// TIA Portal project "GR36_BP_PSElevator" (V17)

(* hardware
DEVICE "ET 200SP station_1"  ET 200SP-Station
   slot 0: "Rack_0"  Rack  6ES5 710-8MAx1
   slot 1: "PLC_1"  CPU 1510SP-1 PN  6ES7 510-1DJ01-0AB0  V2.1
      slot 32768: "PROFINET interface_1"  X1
   slot 2: "DI 8x24VDC HF_1"  DI 8x24VDC HF  6ES7 131-6BF00-0CA0  V2.0
      slot 1: "DI 8x24VDC HF_1"  DI 8x24VDC HF
   slot 3: "DI 8x24VDC BA_1"  DI 8x24VDC BA  6ES7 131-6BF00-0AA0  V1.0
      slot 1: "DI 8x24VDC BA_1"  DI 8x24VDC BA
   slot 4: "DQ 8x24VDC/0.5A ST_1"  DQ 8x24VDC/0.5A ST  6ES7 132-6BF00-0BA0  V1.1
      slot 1: "DQ 8x24VDC/0.5A ST_1"  DQ 8x24VDC/0.5A ST
   slot 5: "AI 2xU/I 2-,4-wire HF_1"  AI 2xU/I 2-,4-wire HF  6ES7 134-6HB00-0CA1  V2.0
      slot 1: "AI 2xU/I 2-,4-wire HF_1"  AI 2xU/I 2-,4-wire HF
   slot 6: "Server module_1"  Server module  6ES7 193-6PA00-0AA0  V1.1
      slot 1: "Server module_1"  Server module
   slot 127: "BA 2xRJ45"  BA 2xRJ45  6ES7 193-6AR00-0AA0  V0.0
      slot 32769: "Port_1"  X1 P1  6ES7 193-6AR00-0AA0
      slot 32770: "Port_2"  X1 P2  6ES7 193-6AR00-0AA0
*)

// ===== PLC "PLC_1"  CPU 1510SP-1 PN =====

VAR_GLOBAL   // PLC tag table "Default tag table"
   "System_Byte" AT %MB70 : Byte;
   "FirstScan" AT %M70.0 : Bool;
   "DiagStatusUpdate" AT %M70.1 : Bool;
   "AlwaysTRUE" AT %M70.2 : Bool;
   "AlwaysFALSE" AT %M70.3 : Bool;
   "Clock_Byte" AT %MB69 : Byte;
   "Clock_10Hz" AT %M69.0 : Bool;
   "Clock_5Hz" AT %M69.1 : Bool;
   "Clock_2.5Hz" AT %M69.2 : Bool;
   "Clock_2Hz" AT %M69.3 : Bool;
   "Clock_1.25Hz" AT %M69.4 : Bool;
   "Clock_1Hz" AT %M69.5 : Bool;
   "Clock_0.625Hz" AT %M69.6 : Bool;
   "Clock_0.5Hz" AT %M69.7 : Bool;
END_VAR

VAR_GLOBAL   // PLC tag table "PLC_dq"
   "dq_LedGreen" AT %Q204.0 : Bool;
   "dq_LedRed" AT %Q204.1 : Bool;
   "dq_LedWhite" AT %Q204.2 : Bool;
   "dq_LedBlue" AT %Q204.3 : Bool;
END_VAR

VAR_GLOBAL   // PLC tag table "PLC_di"
   "di_StartButton" AT %I202.0 : Bool;
   "di_StopButton" AT %I202.1 : Bool;
   "di_Selector" AT %I202.2 : Bool;
   "di_Reset" AT %I202.3 : Bool;
   "di_SwitchForward" AT %I201.0 : Bool;
   "di_SwitchBackward" AT %I201.1 : Bool;
   "di_SwitchBay1" AT %I201.2 : Bool;
   "di_SwitchBay2" AT %I201.3 : Bool;
END_VAR

VAR_GLOBAL   // PLC tag table "FactoryIO_dq"
   "dq_M1" AT %Q7.0 : Bool;
   "dq_M2" AT %Q7.1 : Bool;
   "dq_M3" AT %Q7.2 : Bool;
   "dq_Turntable_1_Turn" AT %Q7.3 : Bool;
   "dq_Turntable_1_Roll+" AT %Q7.4 : Bool;
   "dq_Turntable_1_Roll-" AT %Q7.5 : Bool;
   "dq_Elevator_1_Up" AT %Q8.0 : Bool;
   "dq_Elevator_1_Down" AT %Q8.1 : Bool;
   "dq_Elevator_1_Slow" AT %Q8.2 : Bool;
   "dq_M5" AT %Q8.3 : Bool;
   "dq_M6" AT %Q8.4 : Bool;
   "dq_M4_Elevator_1_+" AT %Q7.6 : Bool;
   "dq_M4_Elevator_1_-" AT %Q7.7 : Bool;
END_VAR

VAR_GLOBAL   // PLC tag table "FactoryIO_di"
   "di_B1" AT %I7.0 : Bool;
   "di_B3_Exit" AT %I7.1 : Bool;
   "di_B5_Exit" AT %I7.2 : Bool;
   "di_B6_Exit" AT %I7.3 : Bool;
   "di_B3_Entry" AT %I7.4 : Bool;
   "di_B5_Entry" AT %I7.5 : Bool;
   "di_B6_Entry" AT %I7.6 : Bool;
   "di_Elevator_1_LeftLimit" AT %I7.7 : Bool;
   "di_Elevator_1_RightLimit" AT %I8.0 : Bool;
   "di_HightSensor_Lift_0" AT %I8.1 : Bool;
   "di_HightSensor_Lift_1" AT %I8.2 : Bool;
   "di_LowSensor_Lift_0" AT %I8.3 : Bool;
   "di_LowSensor_Lift_1" AT %I8.4 : Bool;
   "di_M3_Encoder_Signal_A" AT %I8.5 : Bool;
   "di_M3_Encoder_Signal_B" AT %I8.6 : Bool;
   "di_Turntable_1_Limit_0" AT %I8.7 : Bool;
   "di_Turntable_1_Limit_90" AT %I9.0 : Bool;
   "di_Turntable_1_BackLimit" AT %I9.1 : Bool;
   "di_Turntable_1_FrontLimit" AT %I9.2 : Bool;
   "di_FactoryIO_Running" AT %I9.7 : Bool;
END_VAR

TYPE "edge_detection"
   STRUCT
      OneShoot_Positive : Bool;
      OneShoot_Negative : Bool;
      memory : Struct
         PreviousState_Positive : Bool;
         PreviousState_Negative : Bool;
      END_STRUCT;
   END_STRUCT;
END_TYPE

DATA_BLOCK "db_output"   // DB1
{ S7_Optimized_Access := 'TRUE' }
VERSION : 0.1
   VAR
      M1_Auto_Forward : Bool;
      M2_Auto_Forward : Bool;
      M3_Auto_Forward : Bool;
      "turntable_1_roll_Auto_-" : Bool;
      "turntable_1_roll_Auto_+" : Bool;
      "M4_elevator_1_Auto_+" : Bool;
      "M4_elevator_1_Auto_-" : Bool;
      elevator_1_Auto_Up : Bool;
      elevator_1_Auto_Down : Bool;
      elevator_1_Auto_Slow : Bool;
      M6_Auto_Forward : Bool;
   END_VAR
BEGIN
END_DATA_BLOCK

DATA_BLOCK "db_turntable"   // DB2
{ S7_Optimized_Access := 'TRUE' }
VERSION : 0.1
   VAR
      isOccupied : Bool;
      isM1PackageReady : Bool;
      isM2PackageReady : Bool;
      isM1PackageTransported2Turntable : Bool;
   END_VAR
BEGIN
END_DATA_BLOCK

DATA_BLOCK "db_mode"   // DB3
{ S7_Optimized_Access := 'TRUE' }
VERSION : 0.1
   VAR
      GlobalError : Bool;
      Auto : Bool;
   END_VAR
BEGIN
END_DATA_BLOCK

DATA_BLOCK "db_error"   // DB4
{ S7_Optimized_Access := 'TRUE' }
VERSION : 0.1
   VAR
      er_1 : Bool;
   END_VAR
BEGIN
END_DATA_BLOCK

DATA_BLOCK "db_edge"   // DB5
{ S7_Optimized_Access := 'TRUE' }
VERSION : 0.1
   VAR
      Elevator_1_RightLimit : "edge_detection";
      Elevator_1_LeftLimit : "edge_detection";
      B1 : "edge_detection";
      Turntable_1_BackLimit : "edge_detection";
      Turntable_1_FrontLimit : "edge_detection";
      B3_Entry : "edge_detection";
      B3_End : "edge_detection";
      Lift_1_Height : "edge_detection";
      Lift_1_Low : "edge_detection";
      Lift_0_Height : "edge_detection";
      Lift_0_Low : "edge_detection";
      B6_Entry : "edge_detection";
      B6_Exit : "edge_detection";
      B3_Exit : "edge_detection";
   END_VAR
BEGIN
END_DATA_BLOCK

DATA_BLOCK "db_settings"   // DB6
{ S7_Optimized_Access := 'TRUE' }
VERSION : 0.1
   VAR RETAIN
      M1_ReadyDelay : Time := t#5s;
      M2_ReadyDelay : Time := t#5s;
   END_VAR
BEGIN
END_DATA_BLOCK

DATA_BLOCK "db_elevator"   // DB7
{ S7_Optimized_Access := 'TRUE' }
VERSION : 0.1
   VAR
      isOccupied : Bool;
      slowMode : Bool;
      isLineB3Occupied : Bool;
   END_VAR
BEGIN
END_DATA_BLOCK

FUNCTION "fc_output" : Void   // FC1, LAD
{ S7_Optimized_Access := 'TRUE' }
VERSION : 0.1
BEGIN

REGION Network 1: M1
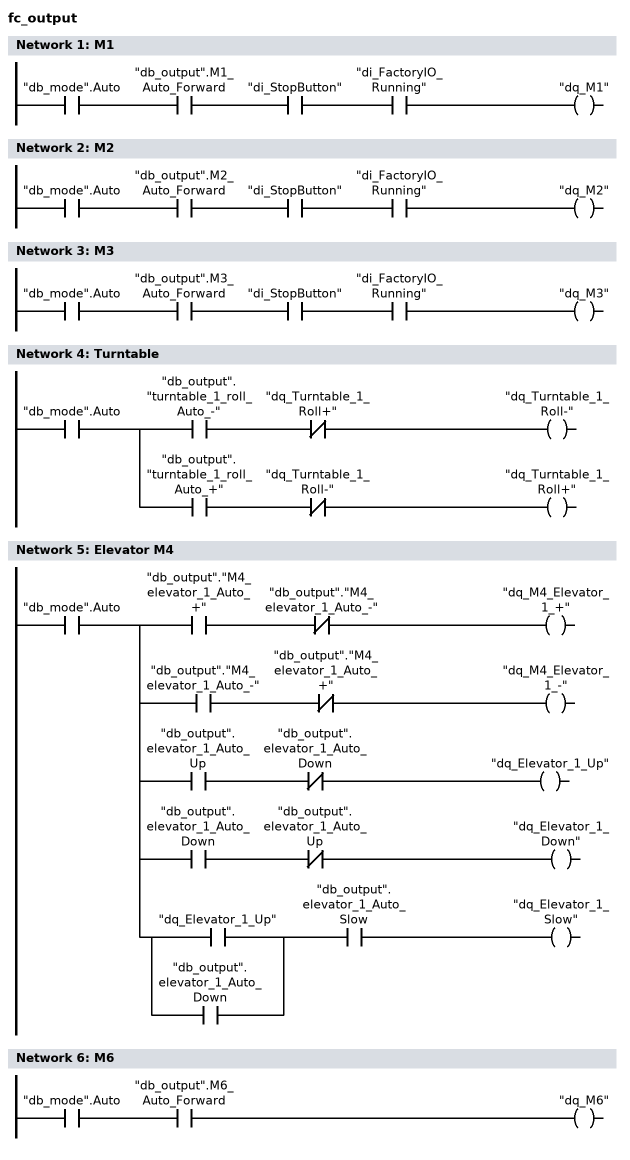
   RUNG wire#powerrail
      Contact( "db_mode".Auto )
      Contact( "db_output".M1_Auto_Forward )
      Contact( "di_StopButton" )
      Contact( "di_FactoryIO_Running" )
      Coil( "dq_M1" )
   END_RUNG
   // the same network as SCL:
   "dq_M1" := "db_mode".Auto AND "db_output".M1_Auto_Forward AND "di_StopButton" AND "di_FactoryIO_Running";
END_REGION

REGION Network 2: M2
   RUNG wire#powerrail
      Contact( "db_mode".Auto )
      Contact( "db_output".M2_Auto_Forward )
      Contact( "di_StopButton" )
      Contact( "di_FactoryIO_Running" )
      Coil( "dq_M2" )
   END_RUNG
   // the same network as SCL:
   "dq_M2" := "db_mode".Auto AND "db_output".M2_Auto_Forward AND "di_StopButton" AND "di_FactoryIO_Running";
END_REGION

REGION Network 3: M3
   RUNG wire#powerrail
      Contact( "db_mode".Auto )
      Contact( "db_output".M3_Auto_Forward )
      Contact( "di_StopButton" )
      Contact( "di_FactoryIO_Running" )
      Coil( "dq_M3" )
   END_RUNG
   // the same network as SCL:
   "dq_M3" := "db_mode".Auto AND "db_output".M3_Auto_Forward AND "di_StopButton" AND "di_FactoryIO_Running";
END_REGION

REGION Network 4: Turntable
   RUNG wire#powerrail
      Contact( "db_mode".Auto )
      wire#w1
      Contact( "db_output"."turntable_1_roll_Auto_-" )
      I_Contact( "dq_Turntable_1_Roll+" )
      Coil( "dq_Turntable_1_Roll-" )
   END_RUNG
   RUNG wire#w1
      Contact( "db_output"."turntable_1_roll_Auto_+" )
      I_Contact( "dq_Turntable_1_Roll-" )
      Coil( "dq_Turntable_1_Roll+" )
   END_RUNG
   // the same network as SCL:
   "dq_Turntable_1_Roll-" := "db_mode".Auto AND "db_output"."turntable_1_roll_Auto_-" AND NOT "dq_Turntable_1_Roll+";
   "dq_Turntable_1_Roll+" := "db_mode".Auto AND "db_output"."turntable_1_roll_Auto_+" AND NOT "dq_Turntable_1_Roll-";
END_REGION

REGION Network 5: Elevator M4
   RUNG wire#powerrail
      Contact( "db_mode".Auto )
      wire#w1
      Contact( "db_output"."M4_elevator_1_Auto_+" )
      I_Contact( "db_output"."M4_elevator_1_Auto_-" )
      Coil( "dq_M4_Elevator_1_+" )
   END_RUNG
   RUNG wire#w1
      Contact( "db_output"."M4_elevator_1_Auto_-" )
      I_Contact( "db_output"."M4_elevator_1_Auto_+" )
      Coil( "dq_M4_Elevator_1_-" )
   END_RUNG
   RUNG wire#w1
      Contact( "db_output".elevator_1_Auto_Up )
      I_Contact( "db_output".elevator_1_Auto_Down )
      Coil( "dq_Elevator_1_Up" )
   END_RUNG
   RUNG wire#w1
      Contact( "db_output".elevator_1_Auto_Down )
      I_Contact( "db_output".elevator_1_Auto_Up )
      Coil( "dq_Elevator_1_Down" )
   END_RUNG
   RUNG wire#w1
      Contact( "dq_Elevator_1_Up" )
      wire#w2
      Contact( "db_output".elevator_1_Auto_Slow )
      Coil( "dq_Elevator_1_Slow" )
   END_RUNG
   RUNG wire#w1
      Contact( "db_output".elevator_1_Auto_Down )
   END_RUNG wire#w2
   // the same network as SCL:
   "dq_M4_Elevator_1_+" := "db_mode".Auto AND "db_output"."M4_elevator_1_Auto_+" AND NOT "db_output"."M4_elevator_1_Auto_-";
   "dq_M4_Elevator_1_-" := "db_mode".Auto AND "db_output"."M4_elevator_1_Auto_-" AND NOT "db_output"."M4_elevator_1_Auto_+";
   "dq_Elevator_1_Up" := "db_mode".Auto AND "db_output".elevator_1_Auto_Up AND NOT "db_output".elevator_1_Auto_Down;
   "dq_Elevator_1_Down" := "db_mode".Auto AND "db_output".elevator_1_Auto_Down AND NOT "db_output".elevator_1_Auto_Up;
   "dq_Elevator_1_Slow" := "db_mode".Auto AND ("dq_Elevator_1_Up" OR "db_output".elevator_1_Auto_Down) AND "db_output".elevator_1_Auto_Slow;
END_REGION

REGION Network 6: M6
   RUNG wire#powerrail
      Contact( "db_mode".Auto )
      Contact( "db_output".M6_Auto_Forward )
      Coil( "dq_M6" )
   END_RUNG
   // the same network as SCL:
   "dq_M6" := "db_mode".Auto AND "db_output".M6_Auto_Forward;
END_REGION
END_FUNCTION

FUNCTION "fc_mode" : Void   // FC2, LAD
{ S7_Optimized_Access := 'TRUE' }
VERSION : 0.1
BEGIN

REGION Network 1: Set auto mode
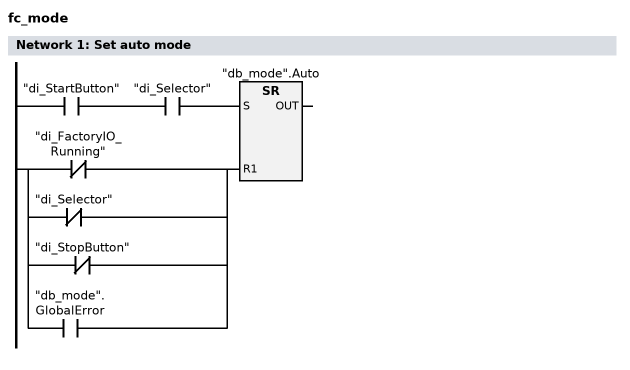
   RUNG wire#powerrail
      Contact( "di_StartButton" )
      Contact( "di_Selector" )
      S_SR(operand := "db_mode".Auto, r1 := wire#w1)
   END_RUNG
   RUNG wire#powerrail
      I_Contact( "di_FactoryIO_Running" )
   END_RUNG wire#w1
   RUNG wire#powerrail
      I_Contact( "di_Selector" )
   END_RUNG wire#w1
   RUNG wire#powerrail
      I_Contact( "di_StopButton" )
   END_RUNG wire#w1
   RUNG wire#powerrail
      Contact( "db_mode".GlobalError )
   END_RUNG wire#w1
   // the same network as SCL:
   IF "di_StartButton" AND "di_Selector" THEN
       "db_mode".Auto := TRUE;   // SR flip-flop
   END_IF;
   IF NOT "di_FactoryIO_Running" OR NOT "di_Selector" OR NOT "di_StopButton" OR "db_mode".GlobalError THEN
       "db_mode".Auto := FALSE;
   END_IF;
END_REGION
END_FUNCTION

FUNCTION "fc_auto" : Void   // FC3, LAD
{ S7_Optimized_Access := 'TRUE' }
VERSION : 0.1
BEGIN

REGION Network 1: M1 Transport the package to the turntable if the turntable is not occupied
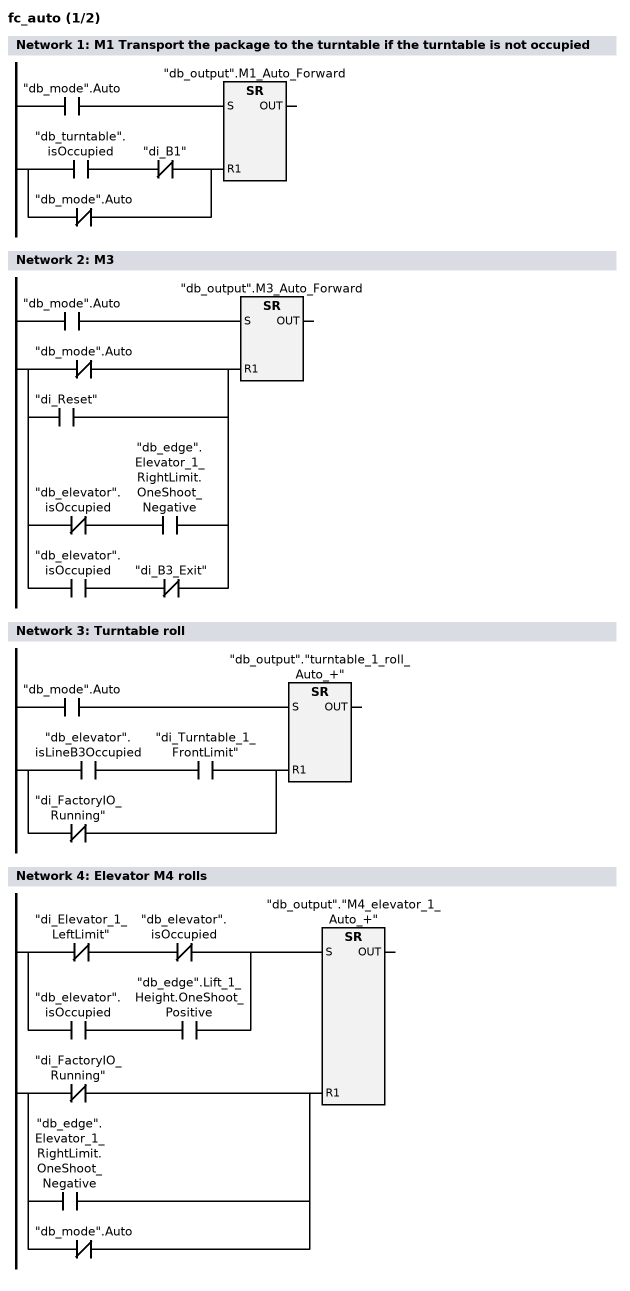
   RUNG wire#powerrail
      Contact( "db_mode".Auto )
      S_SR(operand := "db_output".M1_Auto_Forward, r1 := wire#w1)
   END_RUNG
   RUNG wire#powerrail
      Contact( "db_turntable".isOccupied )
      I_Contact( "di_B1" )
   END_RUNG wire#w1
   RUNG wire#powerrail
      I_Contact( "db_mode".Auto )
   END_RUNG wire#w1
   // the same network as SCL:
   IF "db_mode".Auto THEN
       "db_output".M1_Auto_Forward := TRUE;   // SR flip-flop
   END_IF;
   IF ("db_turntable".isOccupied AND NOT "di_B1") OR NOT "db_mode".Auto THEN
       "db_output".M1_Auto_Forward := FALSE;
   END_IF;
END_REGION

REGION Network 2: M3
   RUNG wire#powerrail
      Contact( "db_mode".Auto )
      S_SR(operand := "db_output".M3_Auto_Forward, r1 := wire#w1)
   END_RUNG
   RUNG wire#powerrail
      I_Contact( "db_mode".Auto )
   END_RUNG wire#w1
   RUNG wire#powerrail
      Contact( "di_Reset" )
   END_RUNG wire#w1
   RUNG wire#powerrail
      I_Contact( "db_elevator".isOccupied )
      Contact( "db_edge".Elevator_1_RightLimit.OneShoot_Negative )
   END_RUNG wire#w1
   RUNG wire#powerrail
      Contact( "db_elevator".isOccupied )
      I_Contact( "di_B3_Exit" )
   END_RUNG wire#w1
   // the same network as SCL:
   IF "db_mode".Auto THEN
       "db_output".M3_Auto_Forward := TRUE;   // SR flip-flop
   END_IF;
   IF NOT "db_mode".Auto OR "di_Reset" OR (NOT "db_elevator".isOccupied AND "db_edge".Elevator_1_RightLimit.OneShoot_Negative) OR ("db_elevator".isOccupied AND NOT "di_B3_Exit") THEN
       "db_output".M3_Auto_Forward := FALSE;
   END_IF;
END_REGION

REGION Network 3: Turntable roll
   RUNG wire#powerrail
      Contact( "db_mode".Auto )
      S_SR(operand := "db_output"."turntable_1_roll_Auto_+", r1 := wire#w1)
   END_RUNG
   RUNG wire#powerrail
      Contact( "db_elevator".isLineB3Occupied )
      Contact( "di_Turntable_1_FrontLimit" )
   END_RUNG wire#w1
   RUNG wire#powerrail
      I_Contact( "di_FactoryIO_Running" )
   END_RUNG wire#w1
   // the same network as SCL:
   IF "db_mode".Auto THEN
       "db_output"."turntable_1_roll_Auto_+" := TRUE;   // SR flip-flop
   END_IF;
   IF ("db_elevator".isLineB3Occupied AND "di_Turntable_1_FrontLimit") OR NOT "di_FactoryIO_Running" THEN
       "db_output"."turntable_1_roll_Auto_+" := FALSE;
   END_IF;
END_REGION

REGION Network 4: Elevator M4 rolls
   RUNG wire#powerrail
      I_Contact( "di_Elevator_1_LeftLimit" )
      I_Contact( "db_elevator".isOccupied )
      wire#w1
      S_SR(operand := "db_output"."M4_elevator_1_Auto_+", r1 := wire#w2)
   END_RUNG
   RUNG wire#powerrail
      Contact( "db_elevator".isOccupied )
      Contact( "db_edge".Lift_1_Height.OneShoot_Positive )
   END_RUNG wire#w1
   RUNG wire#powerrail
      I_Contact( "di_FactoryIO_Running" )
   END_RUNG wire#w2
   RUNG wire#powerrail
      Contact( "db_edge".Elevator_1_RightLimit.OneShoot_Negative )
   END_RUNG wire#w2
   RUNG wire#powerrail
      I_Contact( "db_mode".Auto )
   END_RUNG wire#w2
   // the same network as SCL:
   IF (NOT "di_Elevator_1_LeftLimit" AND NOT "db_elevator".isOccupied) OR ("db_elevator".isOccupied AND "db_edge".Lift_1_Height.OneShoot_Positive) THEN
       "db_output"."M4_elevator_1_Auto_+" := TRUE;   // SR flip-flop
   END_IF;
   IF NOT "di_FactoryIO_Running" OR "db_edge".Elevator_1_RightLimit.OneShoot_Negative OR NOT "db_mode".Auto THEN
       "db_output"."M4_elevator_1_Auto_+" := FALSE;
   END_IF;
END_REGION

REGION Network 5: Elevator lift
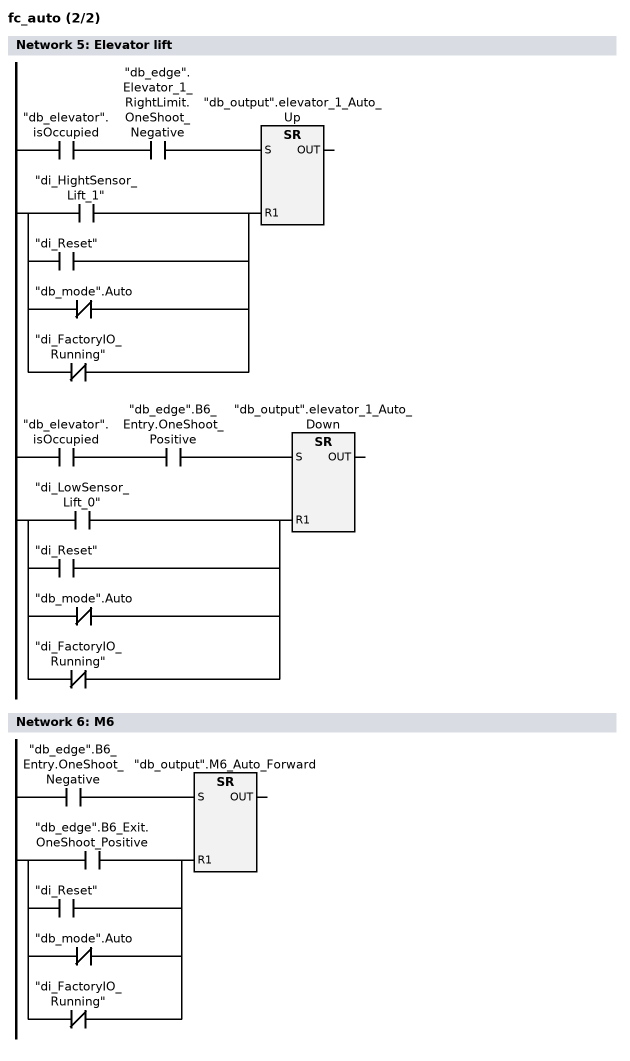
   RUNG wire#powerrail
      Contact( "db_elevator".isOccupied )
      Contact( "db_edge".Elevator_1_RightLimit.OneShoot_Negative )
      S_SR(operand := "db_output".elevator_1_Auto_Up, r1 := wire#w1)
   END_RUNG
   RUNG wire#powerrail
      Contact( "di_HightSensor_Lift_1" )
   END_RUNG wire#w1
   RUNG wire#powerrail
      Contact( "di_Reset" )
   END_RUNG wire#w1
   RUNG wire#powerrail
      I_Contact( "db_mode".Auto )
   END_RUNG wire#w1
   RUNG wire#powerrail
      I_Contact( "di_FactoryIO_Running" )
   END_RUNG wire#w1
   RUNG wire#powerrail
      Contact( "db_elevator".isOccupied )
      Contact( "db_edge".B6_Entry.OneShoot_Positive )
      S_SR(operand := "db_output".elevator_1_Auto_Down, r1 := wire#w2)
   END_RUNG
   RUNG wire#powerrail
      Contact( "di_LowSensor_Lift_0" )
   END_RUNG wire#w2
   RUNG wire#powerrail
      Contact( "di_Reset" )
   END_RUNG wire#w2
   RUNG wire#powerrail
      I_Contact( "db_mode".Auto )
   END_RUNG wire#w2
   RUNG wire#powerrail
      I_Contact( "di_FactoryIO_Running" )
   END_RUNG wire#w2
   // the same network as SCL:
   IF "db_elevator".isOccupied AND "db_edge".Elevator_1_RightLimit.OneShoot_Negative THEN
       "db_output".elevator_1_Auto_Up := TRUE;   // SR flip-flop
   END_IF;
   IF "di_HightSensor_Lift_1" OR "di_Reset" OR NOT "db_mode".Auto OR NOT "di_FactoryIO_Running" THEN
       "db_output".elevator_1_Auto_Up := FALSE;
   END_IF;
   IF "db_elevator".isOccupied AND "db_edge".B6_Entry.OneShoot_Positive THEN
       "db_output".elevator_1_Auto_Down := TRUE;   // SR flip-flop
   END_IF;
   IF "di_LowSensor_Lift_0" OR "di_Reset" OR NOT "db_mode".Auto OR NOT "di_FactoryIO_Running" THEN
       "db_output".elevator_1_Auto_Down := FALSE;
   END_IF;
END_REGION

REGION Network 6: M6
   RUNG wire#powerrail
      Contact( "db_edge".B6_Entry.OneShoot_Negative )
      S_SR(operand := "db_output".M6_Auto_Forward, r1 := wire#w1)
   END_RUNG
   RUNG wire#powerrail
      Contact( "db_edge".B6_Exit.OneShoot_Positive )
   END_RUNG wire#w1
   RUNG wire#powerrail
      Contact( "di_Reset" )
   END_RUNG wire#w1
   RUNG wire#powerrail
      I_Contact( "db_mode".Auto )
   END_RUNG wire#w1
   RUNG wire#powerrail
      I_Contact( "di_FactoryIO_Running" )
   END_RUNG wire#w1
   // the same network as SCL:
   IF "db_edge".B6_Entry.OneShoot_Negative THEN
       "db_output".M6_Auto_Forward := TRUE;   // SR flip-flop
   END_IF;
   IF "db_edge".B6_Exit.OneShoot_Positive OR "di_Reset" OR NOT "db_mode".Auto OR NOT "di_FactoryIO_Running" THEN
       "db_output".M6_Auto_Forward := FALSE;
   END_IF;
END_REGION
END_FUNCTION

FUNCTION "fc_turntable" : Void   // FC4, LAD
{ S7_Optimized_Access := 'TRUE' }
VERSION : 0.1
BEGIN

REGION Network 1: Set when turn table is occupied
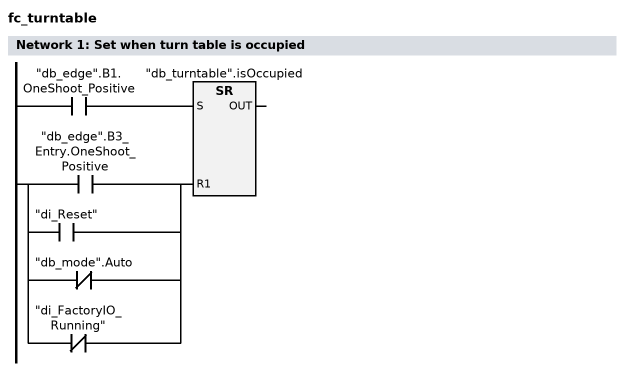
   RUNG wire#powerrail
      Contact( "db_edge".B1.OneShoot_Positive )
      S_SR(operand := "db_turntable".isOccupied, r1 := wire#w1)
   END_RUNG
   RUNG wire#powerrail
      Contact( "db_edge".B3_Entry.OneShoot_Positive )
   END_RUNG wire#w1
   RUNG wire#powerrail
      Contact( "di_Reset" )
   END_RUNG wire#w1
   RUNG wire#powerrail
      I_Contact( "db_mode".Auto )
   END_RUNG wire#w1
   RUNG wire#powerrail
      I_Contact( "di_FactoryIO_Running" )
   END_RUNG wire#w1
   // the same network as SCL:
   IF "db_edge".B1.OneShoot_Positive THEN
       "db_turntable".isOccupied := TRUE;   // SR flip-flop
   END_IF;
   IF "db_edge".B3_Entry.OneShoot_Positive OR "di_Reset" OR NOT "db_mode".Auto OR NOT "di_FactoryIO_Running" THEN
       "db_turntable".isOccupied := FALSE;
   END_IF;
END_REGION
END_FUNCTION

FUNCTION "fc_edge" : Void   // FC5, LAD
{ S7_Optimized_Access := 'TRUE' }
VERSION : 0.1
   VAR_TEMP   // added for the SCL form of the ladder/FBD networks
      _w1 : Bool;
      _w2 : Bool;
      _w3 : Bool;
      _w4 : Bool;
   END_VAR
BEGIN

REGION Network 1: Turntable 1
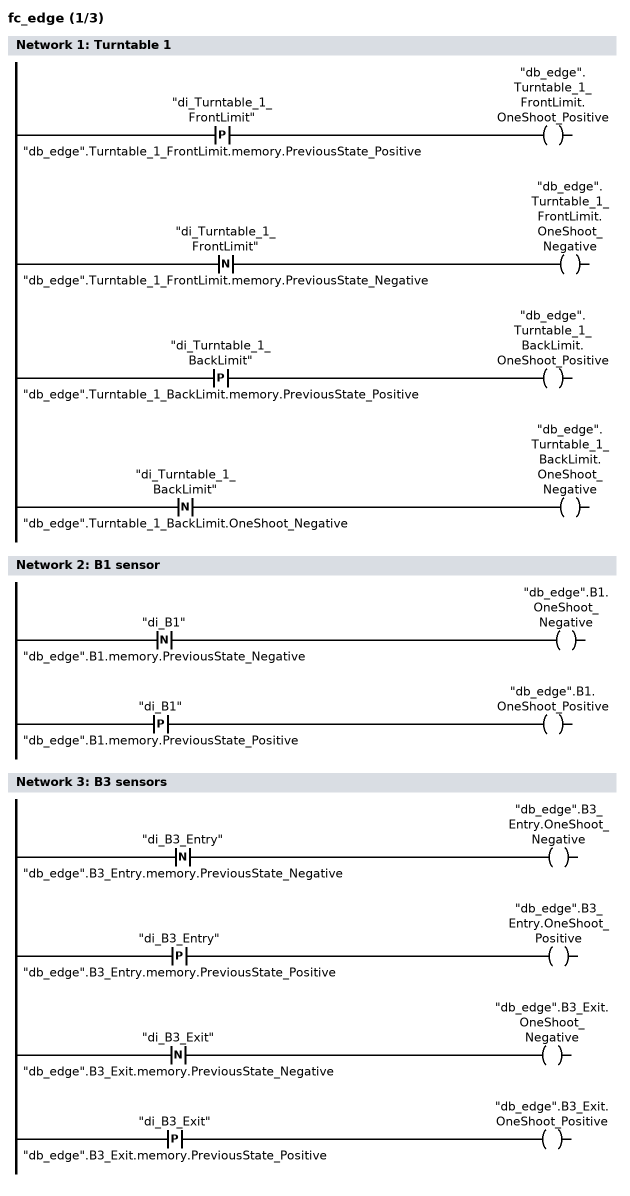
   RUNG wire#powerrail
      P_Contact(operand := "di_Turntable_1_FrontLimit", bit := "db_edge".Turntable_1_FrontLimit.memory.PreviousState_Positive)
      Coil( "db_edge".Turntable_1_FrontLimit.OneShoot_Positive )
   END_RUNG
   RUNG wire#powerrail
      N_Contact(operand := "di_Turntable_1_FrontLimit", bit := "db_edge".Turntable_1_FrontLimit.memory.PreviousState_Negative)
      Coil( "db_edge".Turntable_1_FrontLimit.OneShoot_Negative )
   END_RUNG
   RUNG wire#powerrail
      P_Contact(operand := "di_Turntable_1_BackLimit", bit := "db_edge".Turntable_1_BackLimit.memory.PreviousState_Positive)
      Coil( "db_edge".Turntable_1_BackLimit.OneShoot_Positive )
   END_RUNG
   RUNG wire#powerrail
      N_Contact(operand := "di_Turntable_1_BackLimit", bit := "db_edge".Turntable_1_BackLimit.OneShoot_Negative)
      Coil( "db_edge".Turntable_1_BackLimit.OneShoot_Negative )
   END_RUNG
   // the same network as SCL:
   #_w1 := "di_Turntable_1_FrontLimit" AND NOT "db_edge".Turntable_1_FrontLimit.memory.PreviousState_Positive;   // rising edge of "di_Turntable_1_FrontLimit"
   "db_edge".Turntable_1_FrontLimit.memory.PreviousState_Positive := "di_Turntable_1_FrontLimit";
   "db_edge".Turntable_1_FrontLimit.OneShoot_Positive := #_w1;
   #_w2 := NOT "di_Turntable_1_FrontLimit" AND "db_edge".Turntable_1_FrontLimit.memory.PreviousState_Negative;   // falling edge of "di_Turntable_1_FrontLimit"
   "db_edge".Turntable_1_FrontLimit.memory.PreviousState_Negative := "di_Turntable_1_FrontLimit";
   "db_edge".Turntable_1_FrontLimit.OneShoot_Negative := #_w2;
   #_w3 := "di_Turntable_1_BackLimit" AND NOT "db_edge".Turntable_1_BackLimit.memory.PreviousState_Positive;   // rising edge of "di_Turntable_1_BackLimit"
   "db_edge".Turntable_1_BackLimit.memory.PreviousState_Positive := "di_Turntable_1_BackLimit";
   "db_edge".Turntable_1_BackLimit.OneShoot_Positive := #_w3;
   #_w4 := NOT "di_Turntable_1_BackLimit" AND "db_edge".Turntable_1_BackLimit.OneShoot_Negative;   // falling edge of "di_Turntable_1_BackLimit"
   "db_edge".Turntable_1_BackLimit.OneShoot_Negative := "di_Turntable_1_BackLimit";
   "db_edge".Turntable_1_BackLimit.OneShoot_Negative := #_w4;
END_REGION

REGION Network 2: B1 sensor
   RUNG wire#powerrail
      N_Contact(operand := "di_B1", bit := "db_edge".B1.memory.PreviousState_Negative)
      Coil( "db_edge".B1.OneShoot_Negative )
   END_RUNG
   RUNG wire#powerrail
      P_Contact(operand := "di_B1", bit := "db_edge".B1.memory.PreviousState_Positive)
      Coil( "db_edge".B1.OneShoot_Positive )
   END_RUNG
   // the same network as SCL:
   #_w1 := NOT "di_B1" AND "db_edge".B1.memory.PreviousState_Negative;   // falling edge of "di_B1"
   "db_edge".B1.memory.PreviousState_Negative := "di_B1";
   "db_edge".B1.OneShoot_Negative := #_w1;
   #_w2 := "di_B1" AND NOT "db_edge".B1.memory.PreviousState_Positive;   // rising edge of "di_B1"
   "db_edge".B1.memory.PreviousState_Positive := "di_B1";
   "db_edge".B1.OneShoot_Positive := #_w2;
END_REGION

REGION Network 3: B3 sensors
   RUNG wire#powerrail
      N_Contact(operand := "di_B3_Entry", bit := "db_edge".B3_Entry.memory.PreviousState_Negative)
      Coil( "db_edge".B3_Entry.OneShoot_Negative )
   END_RUNG
   RUNG wire#powerrail
      P_Contact(operand := "di_B3_Entry", bit := "db_edge".B3_Entry.memory.PreviousState_Positive)
      Coil( "db_edge".B3_Entry.OneShoot_Positive )
   END_RUNG
   RUNG wire#powerrail
      N_Contact(operand := "di_B3_Exit", bit := "db_edge".B3_Exit.memory.PreviousState_Negative)
      Coil( "db_edge".B3_Exit.OneShoot_Negative )
   END_RUNG
   RUNG wire#powerrail
      P_Contact(operand := "di_B3_Exit", bit := "db_edge".B3_Exit.memory.PreviousState_Positive)
      Coil( "db_edge".B3_Exit.OneShoot_Positive )
   END_RUNG
   // the same network as SCL:
   #_w1 := NOT "di_B3_Entry" AND "db_edge".B3_Entry.memory.PreviousState_Negative;   // falling edge of "di_B3_Entry"
   "db_edge".B3_Entry.memory.PreviousState_Negative := "di_B3_Entry";
   "db_edge".B3_Entry.OneShoot_Negative := #_w1;
   #_w2 := "di_B3_Entry" AND NOT "db_edge".B3_Entry.memory.PreviousState_Positive;   // rising edge of "di_B3_Entry"
   "db_edge".B3_Entry.memory.PreviousState_Positive := "di_B3_Entry";
   "db_edge".B3_Entry.OneShoot_Positive := #_w2;
   #_w3 := NOT "di_B3_Exit" AND "db_edge".B3_Exit.memory.PreviousState_Negative;   // falling edge of "di_B3_Exit"
   "db_edge".B3_Exit.memory.PreviousState_Negative := "di_B3_Exit";
   "db_edge".B3_Exit.OneShoot_Negative := #_w3;
   #_w4 := "di_B3_Exit" AND NOT "db_edge".B3_Exit.memory.PreviousState_Positive;   // rising edge of "di_B3_Exit"
   "db_edge".B3_Exit.memory.PreviousState_Positive := "di_B3_Exit";
   "db_edge".B3_Exit.OneShoot_Positive := #_w4;
END_REGION

REGION Network 4: Elevator 1
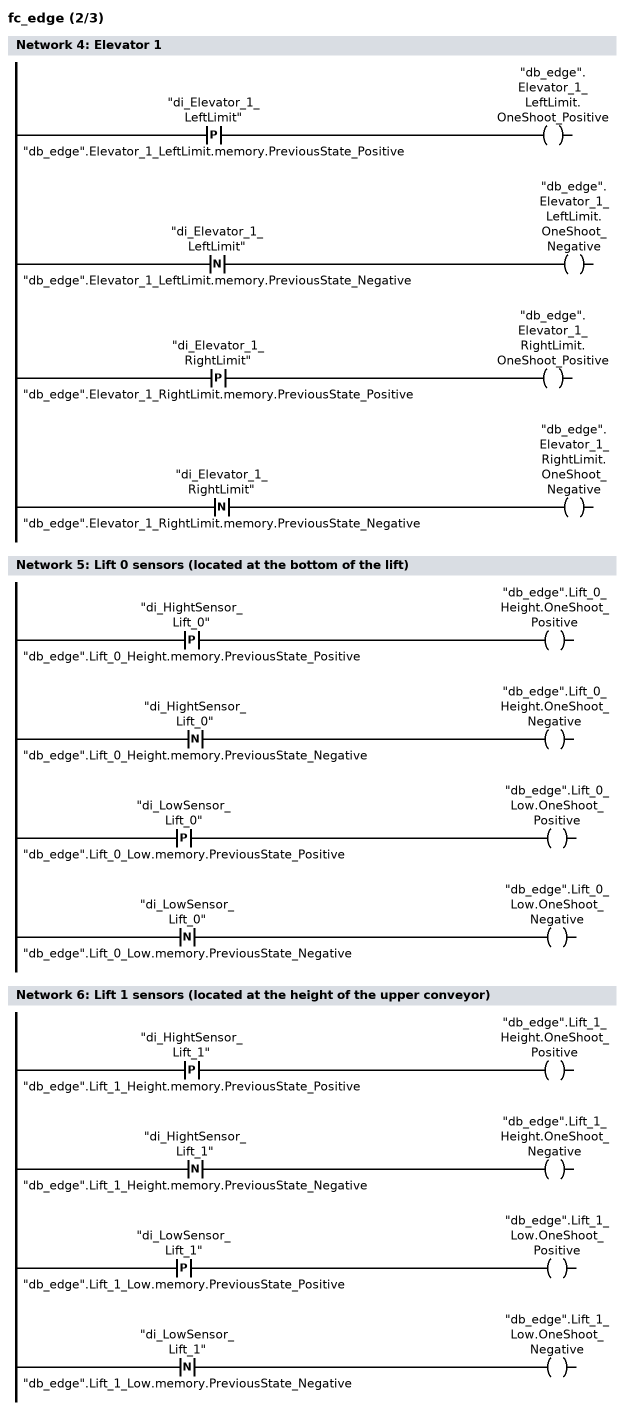
   RUNG wire#powerrail
      P_Contact(operand := "di_Elevator_1_LeftLimit", bit := "db_edge".Elevator_1_LeftLimit.memory.PreviousState_Positive)
      Coil( "db_edge".Elevator_1_LeftLimit.OneShoot_Positive )
   END_RUNG
   RUNG wire#powerrail
      N_Contact(operand := "di_Elevator_1_LeftLimit", bit := "db_edge".Elevator_1_LeftLimit.memory.PreviousState_Negative)
      Coil( "db_edge".Elevator_1_LeftLimit.OneShoot_Negative )
   END_RUNG
   RUNG wire#powerrail
      P_Contact(operand := "di_Elevator_1_RightLimit", bit := "db_edge".Elevator_1_RightLimit.memory.PreviousState_Positive)
      Coil( "db_edge".Elevator_1_RightLimit.OneShoot_Positive )
   END_RUNG
   RUNG wire#powerrail
      N_Contact(operand := "di_Elevator_1_RightLimit", bit := "db_edge".Elevator_1_RightLimit.memory.PreviousState_Negative)
      Coil( "db_edge".Elevator_1_RightLimit.OneShoot_Negative )
   END_RUNG
   // the same network as SCL:
   #_w1 := "di_Elevator_1_LeftLimit" AND NOT "db_edge".Elevator_1_LeftLimit.memory.PreviousState_Positive;   // rising edge of "di_Elevator_1_LeftLimit"
   "db_edge".Elevator_1_LeftLimit.memory.PreviousState_Positive := "di_Elevator_1_LeftLimit";
   "db_edge".Elevator_1_LeftLimit.OneShoot_Positive := #_w1;
   #_w2 := NOT "di_Elevator_1_LeftLimit" AND "db_edge".Elevator_1_LeftLimit.memory.PreviousState_Negative;   // falling edge of "di_Elevator_1_LeftLimit"
   "db_edge".Elevator_1_LeftLimit.memory.PreviousState_Negative := "di_Elevator_1_LeftLimit";
   "db_edge".Elevator_1_LeftLimit.OneShoot_Negative := #_w2;
   #_w3 := "di_Elevator_1_RightLimit" AND NOT "db_edge".Elevator_1_RightLimit.memory.PreviousState_Positive;   // rising edge of "di_Elevator_1_RightLimit"
   "db_edge".Elevator_1_RightLimit.memory.PreviousState_Positive := "di_Elevator_1_RightLimit";
   "db_edge".Elevator_1_RightLimit.OneShoot_Positive := #_w3;
   #_w4 := NOT "di_Elevator_1_RightLimit" AND "db_edge".Elevator_1_RightLimit.memory.PreviousState_Negative;   // falling edge of "di_Elevator_1_RightLimit"
   "db_edge".Elevator_1_RightLimit.memory.PreviousState_Negative := "di_Elevator_1_RightLimit";
   "db_edge".Elevator_1_RightLimit.OneShoot_Negative := #_w4;
END_REGION

REGION Network 5: Lift 0 sensors (located at the bottom of the lift)
   RUNG wire#powerrail
      P_Contact(operand := "di_HightSensor_Lift_0", bit := "db_edge".Lift_0_Height.memory.PreviousState_Positive)
      Coil( "db_edge".Lift_0_Height.OneShoot_Positive )
   END_RUNG
   RUNG wire#powerrail
      N_Contact(operand := "di_HightSensor_Lift_0", bit := "db_edge".Lift_0_Height.memory.PreviousState_Negative)
      Coil( "db_edge".Lift_0_Height.OneShoot_Negative )
   END_RUNG
   RUNG wire#powerrail
      P_Contact(operand := "di_LowSensor_Lift_0", bit := "db_edge".Lift_0_Low.memory.PreviousState_Positive)
      Coil( "db_edge".Lift_0_Low.OneShoot_Positive )
   END_RUNG
   RUNG wire#powerrail
      N_Contact(operand := "di_LowSensor_Lift_0", bit := "db_edge".Lift_0_Low.memory.PreviousState_Negative)
      Coil( "db_edge".Lift_0_Low.OneShoot_Negative )
   END_RUNG
   // the same network as SCL:
   #_w1 := "di_HightSensor_Lift_0" AND NOT "db_edge".Lift_0_Height.memory.PreviousState_Positive;   // rising edge of "di_HightSensor_Lift_0"
   "db_edge".Lift_0_Height.memory.PreviousState_Positive := "di_HightSensor_Lift_0";
   "db_edge".Lift_0_Height.OneShoot_Positive := #_w1;
   #_w2 := NOT "di_HightSensor_Lift_0" AND "db_edge".Lift_0_Height.memory.PreviousState_Negative;   // falling edge of "di_HightSensor_Lift_0"
   "db_edge".Lift_0_Height.memory.PreviousState_Negative := "di_HightSensor_Lift_0";
   "db_edge".Lift_0_Height.OneShoot_Negative := #_w2;
   #_w3 := "di_LowSensor_Lift_0" AND NOT "db_edge".Lift_0_Low.memory.PreviousState_Positive;   // rising edge of "di_LowSensor_Lift_0"
   "db_edge".Lift_0_Low.memory.PreviousState_Positive := "di_LowSensor_Lift_0";
   "db_edge".Lift_0_Low.OneShoot_Positive := #_w3;
   #_w4 := NOT "di_LowSensor_Lift_0" AND "db_edge".Lift_0_Low.memory.PreviousState_Negative;   // falling edge of "di_LowSensor_Lift_0"
   "db_edge".Lift_0_Low.memory.PreviousState_Negative := "di_LowSensor_Lift_0";
   "db_edge".Lift_0_Low.OneShoot_Negative := #_w4;
END_REGION

REGION Network 6: Lift 1 sensors (located at the height of the upper conveyor)
   RUNG wire#powerrail
      P_Contact(operand := "di_HightSensor_Lift_1", bit := "db_edge".Lift_1_Height.memory.PreviousState_Positive)
      Coil( "db_edge".Lift_1_Height.OneShoot_Positive )
   END_RUNG
   RUNG wire#powerrail
      N_Contact(operand := "di_HightSensor_Lift_1", bit := "db_edge".Lift_1_Height.memory.PreviousState_Negative)
      Coil( "db_edge".Lift_1_Height.OneShoot_Negative )
   END_RUNG
   RUNG wire#powerrail
      P_Contact(operand := "di_LowSensor_Lift_1", bit := "db_edge".Lift_1_Low.memory.PreviousState_Positive)
      Coil( "db_edge".Lift_1_Low.OneShoot_Positive )
   END_RUNG
   RUNG wire#powerrail
      N_Contact(operand := "di_LowSensor_Lift_1", bit := "db_edge".Lift_1_Low.memory.PreviousState_Negative)
      Coil( "db_edge".Lift_1_Low.OneShoot_Negative )
   END_RUNG
   // the same network as SCL:
   #_w1 := "di_HightSensor_Lift_1" AND NOT "db_edge".Lift_1_Height.memory.PreviousState_Positive;   // rising edge of "di_HightSensor_Lift_1"
   "db_edge".Lift_1_Height.memory.PreviousState_Positive := "di_HightSensor_Lift_1";
   "db_edge".Lift_1_Height.OneShoot_Positive := #_w1;
   #_w2 := NOT "di_HightSensor_Lift_1" AND "db_edge".Lift_1_Height.memory.PreviousState_Negative;   // falling edge of "di_HightSensor_Lift_1"
   "db_edge".Lift_1_Height.memory.PreviousState_Negative := "di_HightSensor_Lift_1";
   "db_edge".Lift_1_Height.OneShoot_Negative := #_w2;
   #_w3 := "di_LowSensor_Lift_1" AND NOT "db_edge".Lift_1_Low.memory.PreviousState_Positive;   // rising edge of "di_LowSensor_Lift_1"
   "db_edge".Lift_1_Low.memory.PreviousState_Positive := "di_LowSensor_Lift_1";
   "db_edge".Lift_1_Low.OneShoot_Positive := #_w3;
   #_w4 := NOT "di_LowSensor_Lift_1" AND "db_edge".Lift_1_Low.memory.PreviousState_Negative;   // falling edge of "di_LowSensor_Lift_1"
   "db_edge".Lift_1_Low.memory.PreviousState_Negative := "di_LowSensor_Lift_1";
   "db_edge".Lift_1_Low.OneShoot_Negative := #_w4;
END_REGION

REGION Network 7: B6 sensors
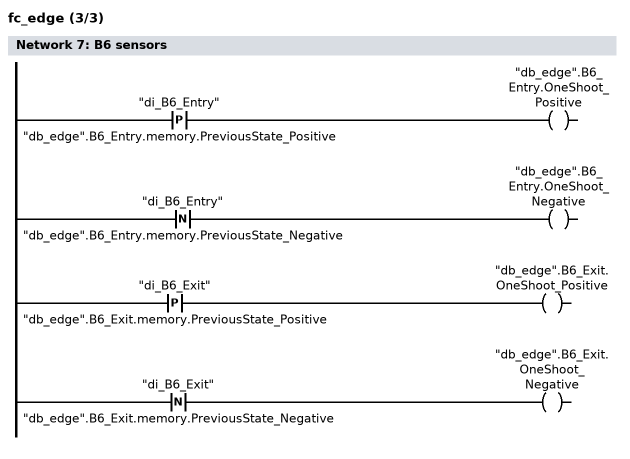
   RUNG wire#powerrail
      P_Contact(operand := "di_B6_Entry", bit := "db_edge".B6_Entry.memory.PreviousState_Positive)
      Coil( "db_edge".B6_Entry.OneShoot_Positive )
   END_RUNG
   RUNG wire#powerrail
      N_Contact(operand := "di_B6_Entry", bit := "db_edge".B6_Entry.memory.PreviousState_Negative)
      Coil( "db_edge".B6_Entry.OneShoot_Negative )
   END_RUNG
   RUNG wire#powerrail
      P_Contact(operand := "di_B6_Exit", bit := "db_edge".B6_Exit.memory.PreviousState_Positive)
      Coil( "db_edge".B6_Exit.OneShoot_Positive )
   END_RUNG
   RUNG wire#powerrail
      N_Contact(operand := "di_B6_Exit", bit := "db_edge".B6_Exit.memory.PreviousState_Negative)
      Coil( "db_edge".B6_Exit.OneShoot_Negative )
   END_RUNG
   // the same network as SCL:
   #_w1 := "di_B6_Entry" AND NOT "db_edge".B6_Entry.memory.PreviousState_Positive;   // rising edge of "di_B6_Entry"
   "db_edge".B6_Entry.memory.PreviousState_Positive := "di_B6_Entry";
   "db_edge".B6_Entry.OneShoot_Positive := #_w1;
   #_w2 := NOT "di_B6_Entry" AND "db_edge".B6_Entry.memory.PreviousState_Negative;   // falling edge of "di_B6_Entry"
   "db_edge".B6_Entry.memory.PreviousState_Negative := "di_B6_Entry";
   "db_edge".B6_Entry.OneShoot_Negative := #_w2;
   #_w3 := "di_B6_Exit" AND NOT "db_edge".B6_Exit.memory.PreviousState_Positive;   // rising edge of "di_B6_Exit"
   "db_edge".B6_Exit.memory.PreviousState_Positive := "di_B6_Exit";
   "db_edge".B6_Exit.OneShoot_Positive := #_w3;
   #_w4 := NOT "di_B6_Exit" AND "db_edge".B6_Exit.memory.PreviousState_Negative;   // falling edge of "di_B6_Exit"
   "db_edge".B6_Exit.memory.PreviousState_Negative := "di_B6_Exit";
   "db_edge".B6_Exit.OneShoot_Negative := #_w4;
END_REGION
END_FUNCTION

FUNCTION "fc_elevator" : Void   // FC6, LAD
{ S7_Optimized_Access := 'TRUE' }
VERSION : 0.1
BEGIN

REGION Network 1: Set when elevator is occupied
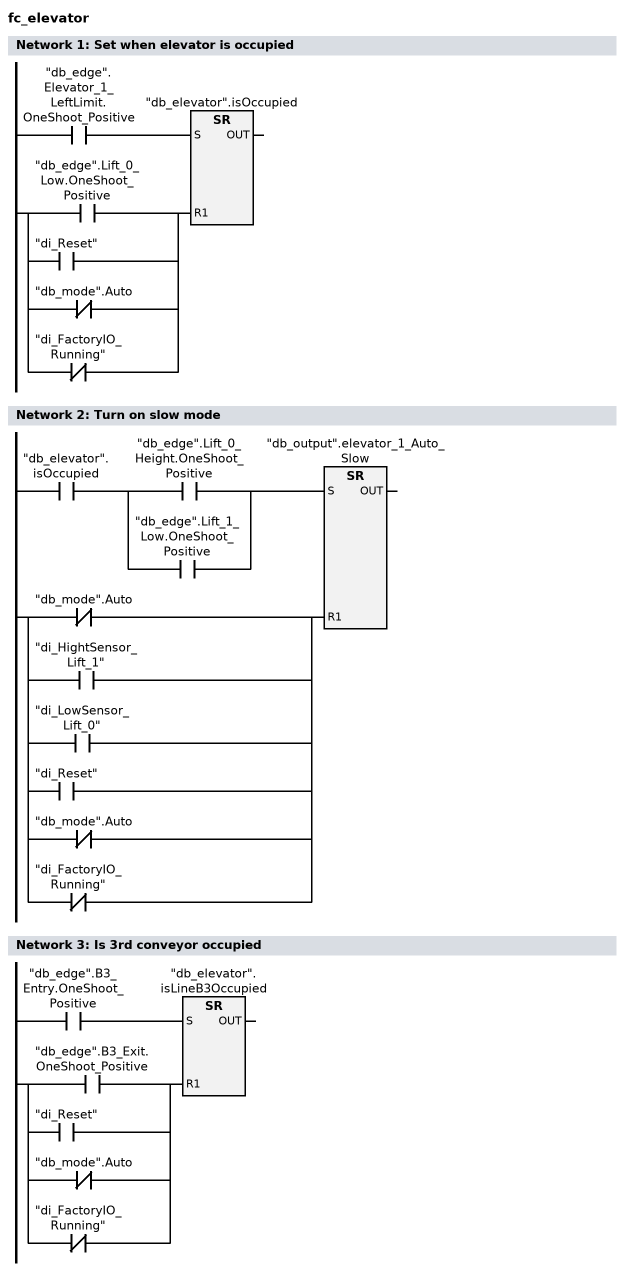
   RUNG wire#powerrail
      Contact( "db_edge".Elevator_1_LeftLimit.OneShoot_Positive )
      S_SR(operand := "db_elevator".isOccupied, r1 := wire#w1)
   END_RUNG
   RUNG wire#powerrail
      Contact( "db_edge".Lift_0_Low.OneShoot_Positive )
   END_RUNG wire#w1
   RUNG wire#powerrail
      Contact( "di_Reset" )
   END_RUNG wire#w1
   RUNG wire#powerrail
      I_Contact( "db_mode".Auto )
   END_RUNG wire#w1
   RUNG wire#powerrail
      I_Contact( "di_FactoryIO_Running" )
   END_RUNG wire#w1
   // the same network as SCL:
   IF "db_edge".Elevator_1_LeftLimit.OneShoot_Positive THEN
       "db_elevator".isOccupied := TRUE;   // SR flip-flop
   END_IF;
   IF "db_edge".Lift_0_Low.OneShoot_Positive OR "di_Reset" OR NOT "db_mode".Auto OR NOT "di_FactoryIO_Running" THEN
       "db_elevator".isOccupied := FALSE;
   END_IF;
END_REGION

REGION Network 2: Turn on slow mode
   RUNG wire#powerrail
      Contact( "db_elevator".isOccupied )
      wire#w1
      Contact( "db_edge".Lift_0_Height.OneShoot_Positive )
      wire#w2
      S_SR(operand := "db_output".elevator_1_Auto_Slow, r1 := wire#w3)
   END_RUNG
   RUNG wire#w1
      Contact( "db_edge".Lift_1_Low.OneShoot_Positive )
   END_RUNG wire#w2
   RUNG wire#powerrail
      I_Contact( "db_mode".Auto )
   END_RUNG wire#w3
   RUNG wire#powerrail
      Contact( "di_HightSensor_Lift_1" )
   END_RUNG wire#w3
   RUNG wire#powerrail
      Contact( "di_LowSensor_Lift_0" )
   END_RUNG wire#w3
   RUNG wire#powerrail
      Contact( "di_Reset" )
   END_RUNG wire#w3
   RUNG wire#powerrail
      I_Contact( "db_mode".Auto )
   END_RUNG wire#w3
   RUNG wire#powerrail
      I_Contact( "di_FactoryIO_Running" )
   END_RUNG wire#w3
   // the same network as SCL:
   IF "db_elevator".isOccupied AND ("db_edge".Lift_0_Height.OneShoot_Positive OR "db_edge".Lift_1_Low.OneShoot_Positive) THEN
       "db_output".elevator_1_Auto_Slow := TRUE;   // SR flip-flop
   END_IF;
   IF NOT "db_mode".Auto OR "di_HightSensor_Lift_1" OR "di_LowSensor_Lift_0" OR "di_Reset" OR NOT "db_mode".Auto OR NOT "di_FactoryIO_Running" THEN
       "db_output".elevator_1_Auto_Slow := FALSE;
   END_IF;
END_REGION

REGION Network 3: Is 3rd conveyor occupied
   RUNG wire#powerrail
      Contact( "db_edge".B3_Entry.OneShoot_Positive )
      S_SR(operand := "db_elevator".isLineB3Occupied, r1 := wire#w1)
   END_RUNG
   RUNG wire#powerrail
      Contact( "db_edge".B3_Exit.OneShoot_Positive )
   END_RUNG wire#w1
   RUNG wire#powerrail
      Contact( "di_Reset" )
   END_RUNG wire#w1
   RUNG wire#powerrail
      I_Contact( "db_mode".Auto )
   END_RUNG wire#w1
   RUNG wire#powerrail
      I_Contact( "di_FactoryIO_Running" )
   END_RUNG wire#w1
   // the same network as SCL:
   IF "db_edge".B3_Entry.OneShoot_Positive THEN
       "db_elevator".isLineB3Occupied := TRUE;   // SR flip-flop
   END_IF;
   IF "db_edge".B3_Exit.OneShoot_Positive OR "di_Reset" OR NOT "db_mode".Auto OR NOT "di_FactoryIO_Running" THEN
       "db_elevator".isLineB3Occupied := FALSE;
   END_IF;
END_REGION
END_FUNCTION

ORGANIZATION_BLOCK "Main"   // OB1, LAD, ProgramCycle
TITLE = "Main Program Sweep (Cycle)"
{ S7_Optimized_Access := 'TRUE' }
VERSION : 0.1
   VAR_INPUT
      Initial_Call : Bool;   // Initial call of this OB
      Remanence : Bool;   // =True, if remanent data are available
   END_VAR
BEGIN

REGION Network 1
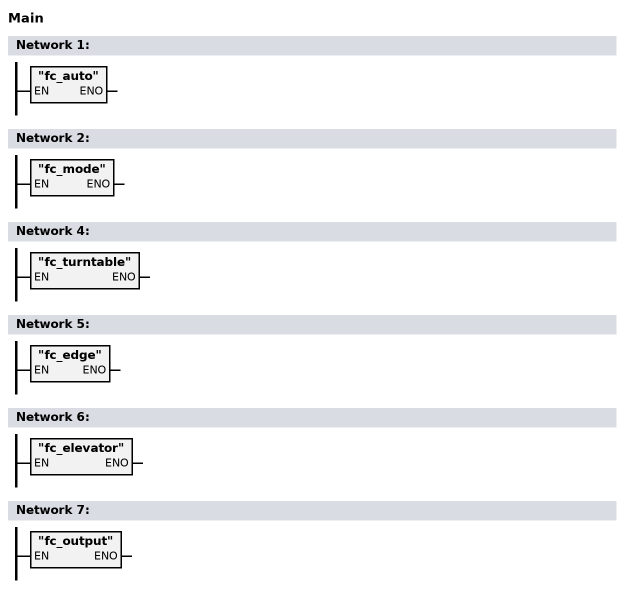
   RUNG wire#powerrail
      "fc_auto"()
   END_RUNG
   // the same network as SCL:
   "fc_auto"();
END_REGION

REGION Network 2
   RUNG wire#powerrail
      "fc_mode"()
   END_RUNG
   // the same network as SCL:
   "fc_mode"();
END_REGION

REGION Network 4
   RUNG wire#powerrail
      "fc_turntable"()
   END_RUNG
   // the same network as SCL:
   "fc_turntable"();
END_REGION

REGION Network 5
   RUNG wire#powerrail
      "fc_edge"()
   END_RUNG
   // the same network as SCL:
   "fc_edge"();
END_REGION

REGION Network 6
   RUNG wire#powerrail
      "fc_elevator"()
   END_RUNG
   // the same network as SCL:
   "fc_elevator"();
END_REGION

REGION Network 7
   RUNG wire#powerrail
      "fc_output"()
   END_RUNG
   // the same network as SCL:
   "fc_output"();
END_REGION
END_ORGANIZATION_BLOCK